// TIA Portal project "SAME PB" (V16)

(* hardware
DEVICE "S7-1200 station_1"  S7-1200 Station
   slot 0: "Rack_0"  S7-1200 Rack  Rack  V1.0
   slot 1: "PLC_1"  CPU 1212C AC/DC/Rly  6ES7 212-1BE40-0XB0  V4.4
*)

// ===== PLC "PLC_1"  CPU 1212C AC/DC/Rly =====

VAR_GLOBAL   // PLC tag table "Default tag table"
   "START" AT %I0.0 : Bool;
   "MOTOR1" AT %Q0.0 : Bool;
   "MOTOR2" AT %Q0.1 : Bool;
   "MARKER" AT %M0.0 : Bool;
   "CM" AT %M0.1 : Bool;
END_VAR

// folder: System blocks/Program resources

DATA_BLOCK "COUNTER"   // DB1
{ S7_Optimized_Access := 'TRUE' }
AUTHOR : Simatic
FAMILY : IEC
NAME : CNTR
VERSION : 1.0
// stored: InstanceOfName IEC_COUNTER
"IEC_COUNTER"
BEGIN
END_DATA_BLOCK

// folder: (top level)

ORGANIZATION_BLOCK "Main"   // OB1, LAD, ProgramCycle
TITLE = "Main Program Sweep (Cycle)"
{ S7_Optimized_Access := 'TRUE' }
VERSION : 0.1
   VAR_INPUT
      Initial_Call : Bool;   // Initial call of this OB
      Remanence : Bool;   // =True, if remanent data are available
   END_VAR
   VAR_TEMP   // added for the SCL form of the ladder/FBD networks
      _w1 : Bool;
   END_VAR
BEGIN

REGION Network 1
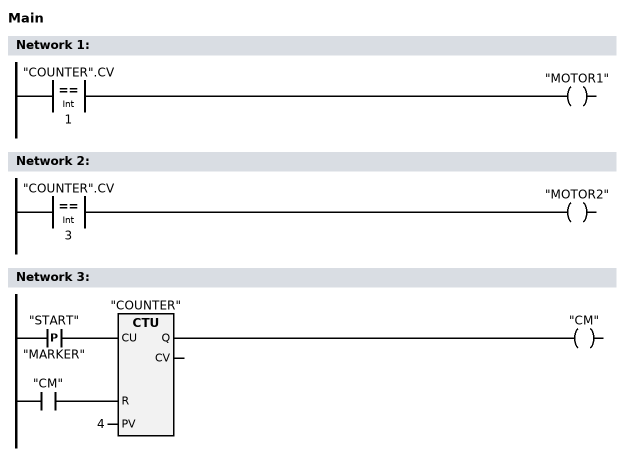
   RUNG wire#powerrail
      { S7_Templates := "SrcType := Int" } EQ_Contact(in1 := "COUNTER".CV, in2 := 1)
      Coil( "MOTOR1" )
   END_RUNG
   // the same network as SCL:
   "MOTOR1" := "COUNTER".CV = 1;
END_REGION

REGION Network 2
   RUNG wire#powerrail
      { S7_Templates := "SrcType := Int" } EQ_Contact(in1 := "COUNTER".CV, in2 := 3)
      Coil( "MOTOR2" )
   END_RUNG
   // the same network as SCL:
   "MOTOR2" := "COUNTER".CV = 3;
END_REGION

REGION Network 3
   #_w1 := "START" AND NOT "MARKER";   // rising edge of "START"
   "MARKER" := "START";
   "COUNTER".CTU(CU := #_w1, R := "CM", PV := 4);
   "CM" := "COUNTER".Q;
END_REGION
END_ORGANIZATION_BLOCK